% RSLogix 500 project PLC LEVEL 2 PROJECT 6.RSS, saved by version 8.30.00.16 %
PROJECT "UNTITLED"    % processor: Bul.1763 MicroLogix 1100 Series B %

PROGRAM FILES
  LAD 2   8 rungs

DATA FILES
  O0 OUTPUT  4 elements
  I1 INPUT  6 elements
  S2 STATUS  66 elements
  B3 BINARY  1 elements
  T4 TIMER  1 elements
  C5 COUNTER  4 elements
  R6 CONTROL  1 elements
  N7 INTEGER  4 elements
  F8 FLOAT  1 elements

LADDER 2
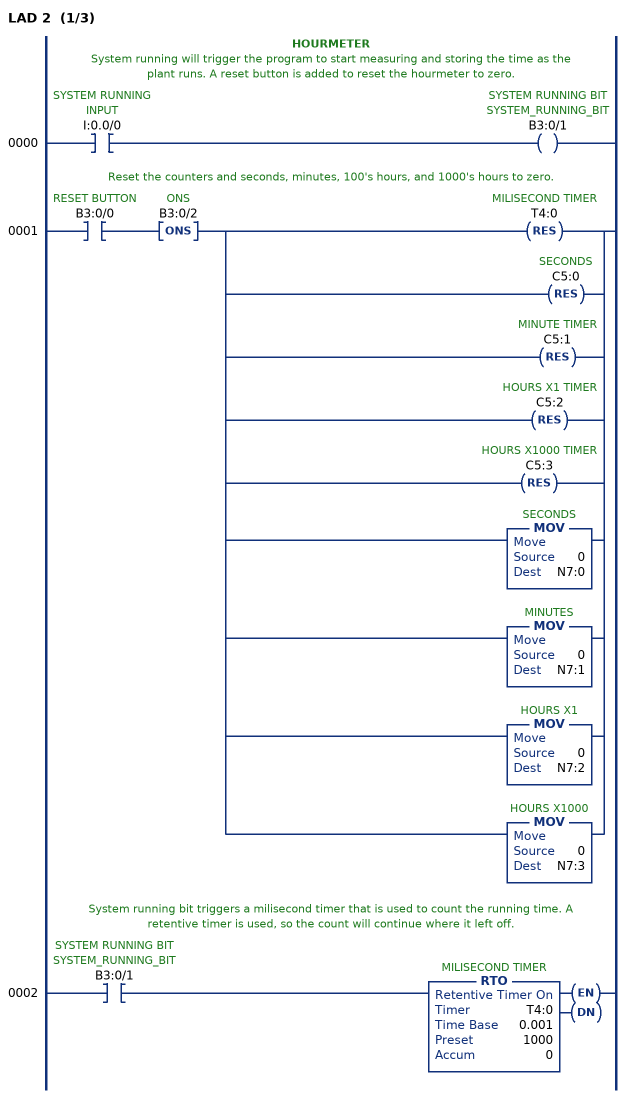
% Rung: 0 %
% TITLE: HOURMETER %
% System running will trigger the program to start measuring and storing the time as the plant runs. A reset button is added to reset the hourmeter to zero. %
SOR XIC I:0.0/0 OTE B3:0/1 EOR
%   I:0.0/0  "SYSTEM RUNNING INPUT" %
%   B3:0/1  SYSTEM_RUNNING_BIT  "SYSTEM RUNNING BIT" %
% Rung: 1 %
% Reset the counters and seconds, minutes, 100's hours, and 1000's hours to zero. %
SOR XIC B3:0/0 ONS B3:0/2 BST RES T4:0 NXB RES C5:0 NXB RES C5:1 NXB RES C5:2 NXB RES C5:3 NXB MOV 0 N7:0 NXB MOV 0 N7:1 NXB MOV 0 N7:2 NXB MOV 0 N7:3 BND EOR
%   B3:0/0  "RESET BUTTON" %
%   B3:0/2  "ONS" %
%   T4:0  "MILISECOND TIMER" %
%   C5:0  "SECONDS" %
%   C5:1  "MINUTE TIMER" %
%   C5:2  "HOURS X1 TIMER" %
%   C5:3  "HOURS X1000 TIMER" %
%   N7:0  "SECONDS" %
%   N7:1  "MINUTES" %
%   N7:2  "HOURS X1" %
%   N7:3  "HOURS X1000" %
% Rung: 2 %
% System running bit triggers a milisecond timer that is used to count the running time. A retentive timer is used, so the count will continue where it left off. %
SOR XIC B3:0/1 RTO T4:0 0.001 1000 0 EOR
%   B3:0/1  SYSTEM_RUNNING_BIT  "SYSTEM RUNNING BIT" %
%   T4:0  "MILISECOND TIMER" %

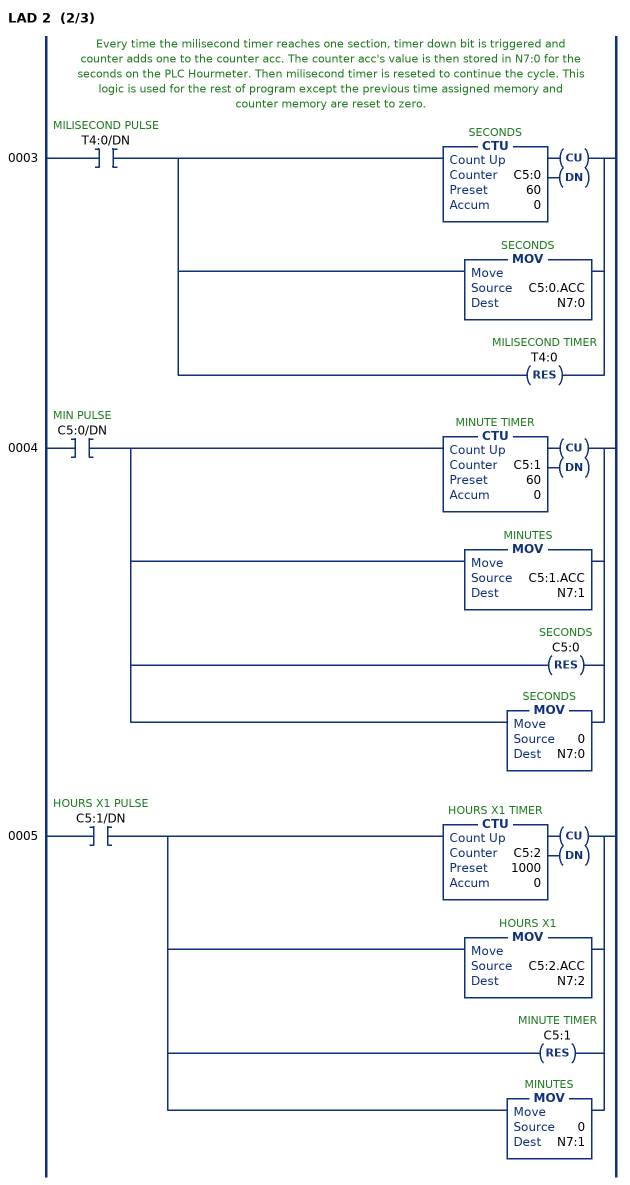
% Rung: 3 %
% Every time the milisecond timer reaches one section, timer down bit is triggered and counter adds one to the counter acc. The counter acc's value is then stored in N7:0 for the seconds on the PLC Hourmeter. Then milisecond timer is reseted to continue the cycle. This logic is used for the rest of program except the previous time assigned memory and counter memory are reset to zero. %
SOR XIC T4:0/DN BST CTU C5:0 60 0 NXB MOV C5:0.ACC N7:0 NXB RES T4:0 BND EOR
%   T4:0/DN  "MILISECOND PULSE" %
%   C5:0  "SECONDS" %
%   C5:0.ACC  "MINUTES" %
%   N7:0  "SECONDS" %
%   T4:0  "MILISECOND TIMER" %
% Rung: 4 %
SOR XIC C5:0/DN BST CTU C5:1 60 0 NXB MOV C5:1.ACC N7:1 NXB RES C5:0 NXB MOV 0 N7:0 BND EOR
%   C5:0/DN  "MIN PULSE" %
%   C5:1  "MINUTE TIMER" %
%   C5:1.ACC  "HOURS" %
%   N7:1  "MINUTES" %
%   C5:0  "SECONDS" %
%   N7:0  "SECONDS" %
% Rung: 5 %
SOR XIC C5:1/DN BST CTU C5:2 1000 0 NXB MOV C5:2.ACC N7:2 NXB RES C5:1 NXB MOV 0 N7:1 BND EOR
%   C5:1/DN  "HOURS X1 PULSE" %
%   C5:2  "HOURS X1 TIMER" %
%   C5:2.ACC  "1000 HOURS" %
%   N7:2  "HOURS X1" %
%   C5:1  "MINUTE TIMER" %
%   N7:1  "MINUTES" %

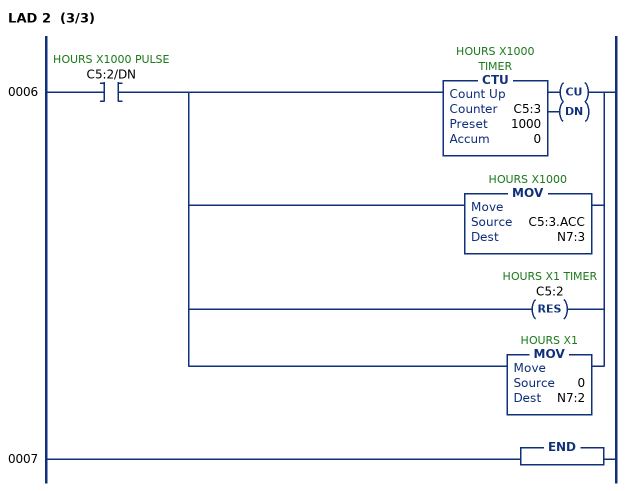
% Rung: 6 %
SOR XIC C5:2/DN BST CTU C5:3 1000 0 NXB MOV C5:3.ACC N7:3 NXB RES C5:2 NXB MOV 0 N7:2 BND EOR
%   C5:2/DN  "HOURS X1000 PULSE" %
%   C5:3  "HOURS X1000 TIMER" %
%   N7:3  "HOURS X1000" %
%   C5:2  "HOURS X1 TIMER" %
%   N7:2  "HOURS X1" %
% Rung: 7 %
SOR END EOR

OTHER DOCUMENTED ADDRESSES
  T4:0.ACC  "SECONDS"
  T4:1  "SECONDS TIMER"

DATA TABLE (non-zero values as saved)
DATA T4
% .PRE .ACC %
% T4:0 % 1000 0
DATA C5
% .PRE .ACC %
% C5:0 % 60 0
% C5:1 % 60 0
% C5:2 % 1000 0
% C5:3 % 1000 0
